(* IEC 61131-3 sources: Intern_HiERN_Testplattform_Hoplyt/Intern_HiERN_Testplattform_PLC/Helpers, 3 files *)

(* ---- BH_AlarmBitTOAlarmArray.st ---- *)
FUNCTION BH_AlarmBitTOAlarmArray : ARRAY[1..8] OF BOOL
VAR_INPUT
	AlarmInfo : SINT;
END_VAR

VAR

END_VAR

		BH_AlarmBitTOAlarmArray[1] := AlarmInfo.0;
		BH_AlarmBitTOAlarmArray[2] := AlarmInfo.1;
		BH_AlarmBitTOAlarmArray[3] := AlarmInfo.2;
		BH_AlarmBitTOAlarmArray[4] := AlarmInfo.3;
		BH_AlarmBitTOAlarmArray[5] := AlarmInfo.4;
		BH_AlarmBitTOAlarmArray[6] := AlarmInfo.5;
		BH_AlarmBitTOAlarmArray[7] := AlarmInfo.6;
		BH_AlarmBitTOAlarmArray[8] := AlarmInfo.7;
;
END_FUNCTION

(* ---- INRANGE.st ---- *)
FUNCTION INRANGE : BOOL
VAR_INPUT
Lower: REAL;
Value: REAL;
Upper: REAL;
END_VAR

VAR

END_VAR

IF Value >= Lower AND Value <= Upper THEN
	INRANGE := TRUE;
ELSE
	INRANGE := FALSE;
END_IF

END_FUNCTION

(* ---- TrimCRLF.st ---- *)
FUNCTION TrimCRLF : STRING
VAR_INPUT
    str : STRING;
END_VAR
VAR
    tmp : STRING;
    L   : INT;
    firstChar, lastChar : STRING;
    CR, LF : STRING;
END_VAR

CR := Util_Chr(BYTE#13);
LF := Util_Chr(BYTE#10);
tmp := str;

(* Leading trim (CR, LF, Space, Tab optional) *)
WHILE LEN(tmp) > 0 DO
    firstChar := LEFT(tmp, 1);
    IF (firstChar = CR) OR (firstChar = LF) OR (firstChar = ' ') OR (firstChar = Util_Chr(Chr := 16#09)) THEN
        tmp := MID(tmp, 2, LEN(tmp) - 1);
    ELSE
        EXIT;
    END_IF;
END_WHILE;

(*  Trailing trim (CR, LF, Space, Tab optional) *)
L := LEN(tmp);
WHILE L > 0 DO
    lastChar := RIGHT(tmp, 1);
    IF (lastChar = CR) OR (lastChar = LF) OR (lastChar = ' ') OR (lastChar = Util_Chr(Chr := 16#09)) THEN
        tmp := LEFT(tmp, L - 1);
        L := L - 1;
    ELSE
        EXIT;
    END_IF;
END_WHILE;

TrimCRLF := tmp;

END_FUNCTION
